PROGRAM MAIN
VAR
END_VAR

END_PROGRAM

(* stored: Version 1.1.0.1
   POU MAIN: Id {b79e520a-676f-4165-bc70-76a19f5b49cd}, SpecialFunc None *)
